ABB RobotStudio station: Second Assignment.rspag

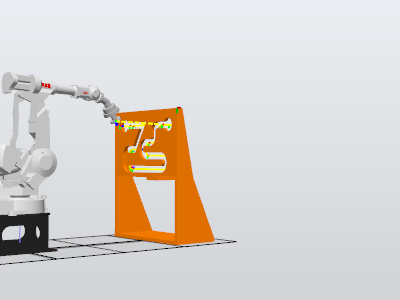
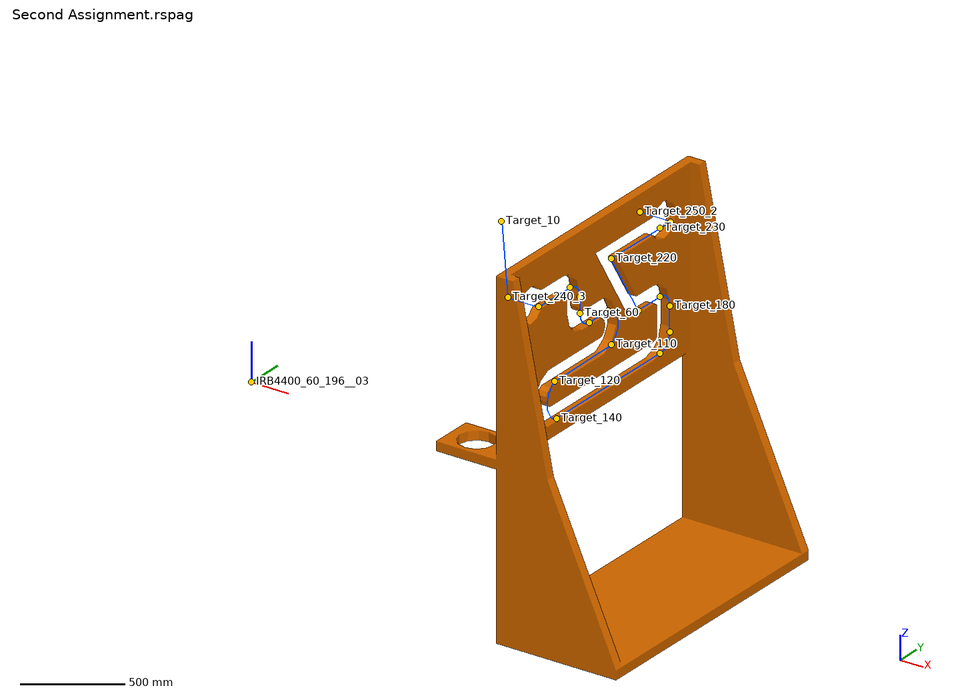
[picture v1: parts stored in the station drawn from their meshes, with robot base, taught points and paths (robot models come from the ABB library and are not in the file)]
--- station ---
Station station (saved by RobotStudio 24.1.10713.1)
Controller Controller3, task T_ROB1: task frame (RAPID world) sits at (0, 0, 500.21) mm in the station
Controller Controller3
  mechanical unit ROB_1: IRB4400_60_196__03, 6 joints, base frame (0, 0, 0) mm
Layout (positions relative to the parent item):
  - IRB4400_60_196__03 [mechanism, from %ABB.RobotStudio.Models.IRB4400%\IRB4400_60_196_G_03.rslib] at (0, 0, 500.21) mm; joint values [0.0465, 0.0523, 0.046, 0.1259, 0.3531, 3.0285] (rad or m)
  - Robotfot_IRB4400 [part, from assignment 2\Robotfot_IRB4400.rslib]
  - Tool [mechanism, from Module 2\Tool.rslib] at (1259.88, 64.75, 2124.37) mm, rotated rx -176.81 ry -67.27 rz 1.91 deg
  - tavla [part] at (2055.32, 720.6, 956.8) mm, rotated rx 90 ry 0 rz -90 deg, size 1600 x 1950 x 1050 mm
  - Part_1 [part] at (2055.32, 720.6, 956.8) mm, rotated rx 90 ry 0 rz -90 deg, size 183.4 x 0 x 50 mm
Attachment: Tool is attached to IRB4400_60_196__03 / Link6
Attachment: Workobject_1 is attached to tavla
Collision set CollisionSet_1: Tool against tavla, near miss 0 m

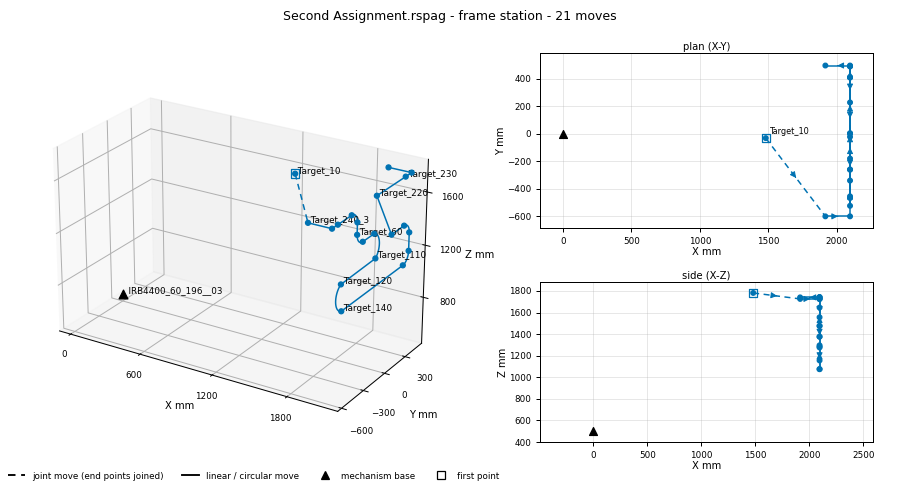
[picture p0: tool path of Second Assignment.rspag in frame station, 21 of 21 moves have a stored position in this frame; points joined in program order, loops and branches not executed]
--- Backups/Controller3/RAPID/TASK1/PROGMOD/CalibData.mod ---
MODULE CalibData
    PERS tooldata Tool:=[TRUE,[[-182.609,0,426.056],[0.958187841,0,-0.286139935,0]],[1,[0,0,1],[1,0,0,0],0,0,0]];
    TASK PERS wobjdata Workobject_1:=[FALSE,TRUE,"",[[2005.321,-829.399720938,1456.591],[0.5,-0.5,0.5,-0.5]],[[0,0,0],[1,0,0,0]]];
ENDMODULE

--- Backups/Controller3/RAPID/TASK1/PROGMOD/Module1.mod ---
MODULE Module1
        CONST robtarget Target_10:=[[-798.050043049,175.415127785,-525.051060351],[0.538949517,-0.371148696,-0.367689139,-0.660747122],[0,-1,1,0],[9E+09,9E+09,9E+09,9E+09,9E+09,9E+09]];
    CONST robtarget Target_20:=[[-306.021800708,230.811964394,89.999518831],[1,0,0,0.000000001],[-1,0,2,0],[9E+09,9E+09,9E+09,9E+09,9E+09,9E+09]];
    CONST robtarget Target_30:=[[-489.41926033,230.811964394,89.999518831],[1,0,0,0.000000001],[-1,0,2,0],[9E+09,9E+09,9E+09,9E+09,9E+09,9E+09]];
    CONST robtarget Target_40:=[[-545.987802787,254.243421862,89.999518831],[1,0,0,0.000000001],[-1,0,2,0],[9E+09,9E+09,9E+09,9E+09,9E+09,9E+09]];
    CONST robtarget Target_50:=[[-569.41926033,310.811964393,89.999518831],[1,0,0,0.000000001],[-1,0,2,0],[9E+09,9E+09,9E+09,9E+09,9E+09,9E+09]];
    CONST robtarget Target_60:=[[-569.41926033,400.811964393,89.999518831],[1,0,0,0.000000001],[-1,0,2,0],[9E+09,9E+09,9E+09,9E+09,9E+09,9E+09]];
    CONST robtarget Target_70:=[[-592.850717797,457.380506852,89.999518831],[1,0,0,0.000000001],[-1,0,2,0],[9E+09,9E+09,9E+09,9E+09,9E+09,9E+09]];
    CONST robtarget Target_80:=[[-649.41926033,480.811964394,89.999518831],[1,0,0,0.000000001],[-1,0,2,0],[9E+09,9E+09,9E+09,9E+09,9E+09,9E+09]];
    CONST robtarget Target_90:=[[-807.406978952,480.811964394,89.999518831],[1,0,0,0.000000001],[0,0,2,0],[9E+09,9E+09,9E+09,9E+09,9E+09,9E+09]];
    CONST robtarget Target_100:=[[-885.138458405,580.811964394,89.999518831],[1,0,0,0.000000001],[0,0,2,0],[9E+09,9E+09,9E+09,9E+09,9E+09,9E+09]];
    CONST robtarget Target_110:=[[-833.882147816,673.227355865,89.999518831],[1,0,0,0.000000001],[0,0,2,0],[9E+09,9E+09,9E+09,9E+09,9E+09,9E+09]];
    CONST robtarget Target_120:=[[-362.535900123,680.811964394,89.999518831],[1,0,0,0.000000001],[-1,0,2,0],[9E+09,9E+09,9E+09,9E+09,9E+09,9E+09]];
    CONST robtarget Target_130:=[[-295.929904216,780.811964394,89.999518831],[1,0,0,0.000000001],[-1,0,2,0],[9E+09,9E+09,9E+09,9E+09,9E+09,9E+09]];
    CONST robtarget Target_140:=[[-374.868021865,882.356636788,89.999518831],[1,0,0,0.000000001],[-1,0,2,0],[9E+09,9E+09,9E+09,9E+09,9E+09,9E+09]];
    CONST robtarget Target_150:=[[-1239.41926033,880.811964394,89.999518831],[1,0,0,0.000000001],[0,0,2,0],[9E+09,9E+09,9E+09,9E+09,9E+09,9E+09]];
    CONST robtarget Target_160:=[[-1295.987802862,857.380506852,89.999518831],[1,0,0,0.000000001],[0,0,2,0],[9E+09,9E+09,9E+09,9E+09,9E+09,9E+09]];
    CONST robtarget Target_170:=[[-1319.41926033,800.811964393,89.999518831],[1,0,0,0.000000001],[0,0,2,0],[9E+09,9E+09,9E+09,9E+09,9E+09,9E+09]];
    CONST robtarget Target_180:=[[-1319.41926033,660.811964393,89.999518831],[1,0,0,0.000000001],[0,0,2,0],[9E+09,9E+09,9E+09,9E+09,9E+09,9E+09]];
    CONST robtarget Target_190:=[[-1295.987802862,604.243421935,89.999518831],[1,0,0,0.000000001],[0,0,2,0],[9E+09,9E+09,9E+09,9E+09,9E+09,9E+09]];
    CONST robtarget Target_200:=[[-1239.41926033,580.811964394,89.999518831],[1,0,0,0.000000001],[0,0,2,0],[9E+09,9E+09,9E+09,9E+09,9E+09,9E+09]];
    CONST robtarget Target_210:=[[-1057.306096355,580.811964393,89.999518831],[1,0,0,0.000000001],[0,0,2,0],[9E+09,9E+09,9E+09,9E+09,9E+09,9E+09]];
    CONST robtarget Target_220:=[[-830.471485674,212.952696239,89.999518831],[1,0,0,0.000000001],[0,0,2,0],[9E+09,9E+09,9E+09,9E+09,9E+09,9E+09]];
    CONST robtarget Target_230:=[[-1239.034176521,216.505554326,89.999518831],[1,0,0,0.000000001],[0,0,2,0],[9E+09,9E+09,9E+09,9E+09,9E+09,9E+09]];
    CONST robtarget Target_240:=[[-229.419720938,230.812241944,90],[1,0,0,0.000000001],[-1,0,2,0],[9E+09,9E+09,9E+09,9E+09,9E+09,9E+09]];
    CONST robtarget Target_250:=[[-1325.636720938,216.505241944,90],[0.996194698,0,0,-0.087155742],[0,0,2,0],[9E+09,9E+09,9E+09,9E+09,9E+09,9E+09]];
    CONST robtarget Target_260:=[[-828.754222431,730.811964394,49.999518831],[0.866025404,0,0,0.5],[0,-2,1,0],[9E+09,9E+09,9E+09,9E+09,9E+09,9E+09]];
    CONST robtarget Target_270:=[[-378.327740435,730.811964394,49.999518831],[0.866025404,0,0,0.5],[-1,-2,1,0],[9E+09,9E+09,9E+09,9E+09,9E+09,9E+09]];
    CONST robtarget Target_280:=[[-378.327740435,730.811964394,-0.000481169],[0.866025404,0,0,0.5],[-1,-2,1,0],[9E+09,9E+09,9E+09,9E+09,9E+09,9E+09]];
    CONST robtarget Target_290:=[[-349.904940542,760.32494624,-0.000481169],[0.866025404,0,0,0.5],[-1,-2,1,0],[9E+09,9E+09,9E+09,9E+09,9E+09,9E+09]];
    CONST robtarget Target_300:=[[-349.904940542,801.298982547,-0.000481169],[0.866025404,0,0,0.5],[-1,-2,1,0],[9E+09,9E+09,9E+09,9E+09,9E+09,9E+09]];
    CONST robtarget Target_310:=[[-378.327740435,830.811964394,-0.000481169],[0.866025404,0,0,0.5],[-1,-2,1,0],[9E+09,9E+09,9E+09,9E+09,9E+09,9E+09]];
    CONST robtarget Target_320:=[[-349.904940542,760.32494624,-0.000481169],[0.866025404,0,0,0.5],[-1,-2,1,0],[9E+09,9E+09,9E+09,9E+09,9E+09,9E+09]];
    CONST robtarget Target_330:=[[-349.904940542,801.298982547,-0.000481169],[0.866025404,0,0,0.5],[-1,-2,1,0],[9E+09,9E+09,9E+09,9E+09,9E+09,9E+09]];
    CONST robtarget Target_340:=[[-378.327740435,830.811964394,-0.000481169],[0.866025404,0,0,0.5],[-1,-2,1,0],[9E+09,9E+09,9E+09,9E+09,9E+09,9E+09]];
    CONST robtarget Target_350:=[[-1239.41926033,830.811964394,-0.000481169],[0.866025404,0,0,0.5],[0,-2,1,0],[9E+09,9E+09,9E+09,9E+09,9E+09,9E+09]];
    CONST robtarget Target_360:=[[-1254.41926033,826.792726507,-0.000481169],[0.866025404,0,0,0.5],[0,-2,1,0],[9E+09,9E+09,9E+09,9E+09,9E+09,9E+09]];
    CONST robtarget Target_370:=[[-1265.400022443,815.811964393,-0.000481169],[0.866025404,0,0,0.5],[0,-2,1,0],[9E+09,9E+09,9E+09,9E+09,9E+09,9E+09]];
    CONST robtarget Target_380:=[[-1269.41926033,800.811964393,-0.000481169],[0.866025404,0,0,0.5],[0,-2,1,0],[9E+09,9E+09,9E+09,9E+09,9E+09,9E+09]];
    CONST robtarget Target_390:=[[-1269.41926033,660.811964393,-0.000481169],[0.866025404,0,0,0.5],[0,-2,0,0],[9E+09,9E+09,9E+09,9E+09,9E+09,9E+09]];
    CONST robtarget Target_400:=[[-1265.400022443,645.811964393,-0.000481169],[0.866025404,0,0,0.5],[0,-2,0,0],[9E+09,9E+09,9E+09,9E+09,9E+09,9E+09]];
    CONST robtarget Target_410:=[[-1254.41926033,634.83120228,-0.000481169],[0.866025404,0,0,0.5],[0,-2,0,0],[9E+09,9E+09,9E+09,9E+09,9E+09,9E+09]];
    CONST robtarget Target_420:=[[-1239.41926033,630.811964394,-0.000481169],[0.866025404,0,0,0.5],[0,-2,0,0],[9E+09,9E+09,9E+09,9E+09,9E+09,9E+09]];
    CONST robtarget Target_430:=[[-1041.532424304,630.811964393,-0.000481169],[0.866025404,0,0,0.5],[0,-2,0,0],[9E+09,9E+09,9E+09,9E+09,9E+09,9E+09]];
    CONST robtarget Target_440:=[[-754.771227196,166.505554326,-0.000481169],[0.866025404,0,0,0.5],[0,-1,0,0],[9E+09,9E+09,9E+09,9E+09,9E+09,9E+09]];
    CONST robtarget Target_450:=[[-1239.034176521,166.505554326,-0.000481169],[0.866025404,0,0,0.5],[0,-1,0,0],[9E+09,9E+09,9E+09,9E+09,9E+09,9E+09]];
    CONST robtarget Target_460:=[[-1280.756798879,127.142290293,-0.000481169],[0.866025404,0,0,0.5],[0,-1,0,0],[9E+09,9E+09,9E+09,9E+09,9E+09,9E+09]];
    CONST robtarget Target_470:=[[-1337.246008312,117.181718551,-0.000481169],[0.866025404,0,0,0.5],[0,-1,0,0],[9E+09,9E+09,9E+09,9E+09,9E+09,9E+09]];
    CONST robtarget Target_480:=[[-1389.915477868,139.901110014,-0.000481169],[0.866025404,0,0,0.5],[0,-1,0,0],[9E+09,9E+09,9E+09,9E+09,9E+09,9E+09]];
    CONST robtarget Target_490:=[[-1421.435668131,187.825231055,-0.000481169],[0.866025404,0,0,0.5],[0,-1,0,0],[9E+09,9E+09,9E+09,9E+09,9E+09,9E+09]];
    CONST robtarget Target_500:=[[-1421.435668131,245.185877597,-0.000481169],[0.866025404,0,0,0.5],[0,-1,0,0],[9E+09,9E+09,9E+09,9E+09,9E+09,9E+09]];
    CONST robtarget Target_510:=[[-1389.915477868,293.109998638,-0.000481169],[0.866025404,0,0,0.5],[0,-1,0,0],[9E+09,9E+09,9E+09,9E+09,9E+09,9E+09]];
    CONST robtarget Target_520:=[[-1337.246008311,315.8293901,-0.000481169],[0.866025404,0,0,0.5],[0,-1,0,0],[9E+09,9E+09,9E+09,9E+09,9E+09,9E+09]];
    CONST robtarget Target_530:=[[-1280.756798879,305.868818358,-0.000481169],[0.866025404,0,0,0.5],[0,-1,0,0],[9E+09,9E+09,9E+09,9E+09,9E+09,9E+09]];
    CONST robtarget Target_540:=[[-1239.034176521,266.505554326,-0.000481169],[0.866025404,0,0,0.5],[0,-1,0,0],[9E+09,9E+09,9E+09,9E+09,9E+09,9E+09]];
    CONST robtarget Target_550:=[[-934.067293463,266.505554325,-0.000481169],[0.866025404,0,0,0.5],[0,-1,0,0],[9E+09,9E+09,9E+09,9E+09,9E+09,9E+09]];
    CONST robtarget Target_560:=[[-934.067293463,266.505554325,49.999518831],[0.866025404,0,0,0.5],[0,-1,0,0],[9E+09,9E+09,9E+09,9E+09,9E+09,9E+09]];
    CONST robtarget Target_570:=[[-1097.306096355,530.811964393,49.999518831],[0.866025404,0,0,0.5],[0,-2,0,0],[9E+09,9E+09,9E+09,9E+09,9E+09,9E+09]];
    CONST robtarget Target_580:=[[-1239.41926033,530.811964394,49.999518831],[0.866025404,0,0,0.5],[0,-1,0,0],[9E+09,9E+09,9E+09,9E+09,9E+09,9E+09]];
    CONST robtarget Target_590:=[[-1304.41926033,548.228661902,49.999518831],[0.866025404,0,0,0.5],[0,-1,0,0],[9E+09,9E+09,9E+09,9E+09,9E+09,9E+09]];
    CONST robtarget Target_600:=[[-1352.002562822,595.811964394,49.999518831],[0.866025404,0,0,0.5],[0,-1,0,0],[9E+09,9E+09,9E+09,9E+09,9E+09,9E+09]];
    CONST robtarget Target_610:=[[-1369.41926033,660.811964393,49.999518831],[0.866025404,0,0,0.5],[0,-2,0,0],[9E+09,9E+09,9E+09,9E+09,9E+09,9E+09]];
    CONST robtarget Target_620:=[[-1369.41926033,800.811964393,49.999518831],[0.866025404,0,0,0.5],[0,-2,1,0],[9E+09,9E+09,9E+09,9E+09,9E+09,9E+09]];
    CONST robtarget Target_630:=[[-1352.002562822,865.811964393,49.999518831],[0.866025404,0,0,0.5],[0,-2,1,0],[9E+09,9E+09,9E+09,9E+09,9E+09,9E+09]];
    CONST robtarget Target_640:=[[-1304.41926033,913.395266885,49.999518831],[0.866025404,0,0,0.5],[0,-2,1,0],[9E+09,9E+09,9E+09,9E+09,9E+09,9E+09]];
    CONST robtarget Target_650:=[[-1239.41926033,930.811964393,49.999518831],[0.866025404,0,0,0.5],[0,-2,1,0],[9E+09,9E+09,9E+09,9E+09,9E+09,9E+09]];
    CONST robtarget Target_660:=[[-362.535900123,930.811964394,49.999518831],[0.866025404,0,0,0.5],[-1,-2,1,0],[9E+09,9E+09,9E+09,9E+09,9E+09,9E+09]];
    CONST robtarget Target_670:=[[-302.218171068,900.212228118,49.999518831],[0.866025404,0,0,0.5],[-1,-2,1,0],[9E+09,9E+09,9E+09,9E+09,9E+09,9E+09]];
    CONST robtarget Target_680:=[[-260.707397504,846.813464306,49.999518831],[0.866025404,0,0,0.5],[-1,-3,1,0],[9E+09,9E+09,9E+09,9E+09,9E+09,9E+09]];
    CONST robtarget Target_690:=[[-245.929904216,780.811964394,49.999518831],[0.866025404,0,0,0.5],[-1,-3,1,0],[9E+09,9E+09,9E+09,9E+09,9E+09,9E+09]];
    CONST robtarget Target_700:=[[-260.707397504,714.810464481,49.999518831],[0.866025404,0,0,0.5],[-1,-3,1,0],[9E+09,9E+09,9E+09,9E+09,9E+09,9E+09]];
    CONST robtarget Target_710:=[[-302.218171068,661.411700669,49.999518831],[0.866025404,0,0,0.5],[-1,-2,1,0],[9E+09,9E+09,9E+09,9E+09,9E+09,9E+09]];
    CONST robtarget Target_720:=[[-362.535900123,630.811964394,49.999518831],[0.866025404,0,0,0.5],[-1,-2,1,0],[9E+09,9E+09,9E+09,9E+09,9E+09,9E+09]];
    CONST robtarget Target_730:=[[-807.406978952,630.811964394,49.999518831],[0.866025404,0,0,0.5],[0,-2,1,0],[9E+09,9E+09,9E+09,9E+09,9E+09,9E+09]];
    CONST robtarget Target_740:=[[-831.811504771,600.334219668,49.999518831],[0.866025404,0,0,0.5],[0,-2,0,0],[9E+09,9E+09,9E+09,9E+09,9E+09,9E+09]];
    CONST robtarget Target_750:=[[-831.811504771,561.289709119,49.999518831],[0.866025404,0,0,0.5],[0,-2,0,0],[9E+09,9E+09,9E+09,9E+09,9E+09,9E+09]];
    CONST robtarget Target_760:=[[-807.406978952,530.811964393,49.999518831],[0.866025404,0,0,0.5],[0,-2,0,0],[9E+09,9E+09,9E+09,9E+09,9E+09,9E+09]];
    CONST robtarget Target_770:=[[-649.41926033,530.811964394,49.999518831],[0.866025404,0,0,0.5],[-1,-2,0,0],[9E+09,9E+09,9E+09,9E+09,9E+09,9E+09]];
    CONST robtarget Target_780:=[[-584.41926033,513.395266885,49.999518831],[0.866025404,0,0,0.5],[-1,-2,0,0],[9E+09,9E+09,9E+09,9E+09,9E+09,9E+09]];
    CONST robtarget Target_790:=[[-536.835957838,465.811964393,49.999518831],[0.866025404,0,0,0.5],[-1,-2,0,0],[9E+09,9E+09,9E+09,9E+09,9E+09,9E+09]];
    CONST robtarget Target_800:=[[-519.41926033,400.811964393,49.999518831],[0.866025404,0,0,0.5],[-1,-1,0,0],[9E+09,9E+09,9E+09,9E+09,9E+09,9E+09]];
    CONST robtarget Target_810:=[[-519.41926033,310.811964393,49.999518831],[0.866025404,0,0,0.5],[-1,-1,0,0],[9E+09,9E+09,9E+09,9E+09,9E+09,9E+09]];
    CONST robtarget Target_820:=[[-515.400022443,295.811964393,49.999518831],[0.866025404,0,0,0.5],[-1,-1,0,0],[9E+09,9E+09,9E+09,9E+09,9E+09,9E+09]];
    CONST robtarget Target_830:=[[-504.41926033,284.83120228,49.999518831],[0.866025404,0,0,0.5],[-1,-1,0,0],[9E+09,9E+09,9E+09,9E+09,9E+09,9E+09]];
    CONST robtarget Target_840:=[[-489.41926033,280.811964393,49.999518831],[0.866025404,0,0,0.5],[-1,-1,0,0],[9E+09,9E+09,9E+09,9E+09,9E+09,9E+09]];
    CONST robtarget Target_850:=[[-306.021800708,280.811964394,49.999518831],[0.866025404,0,0,0.5],[-1,-1,-1,0],[9E+09,9E+09,9E+09,9E+09,9E+09,9E+09]];
    CONST robtarget Target_860:=[[-264.29917835,320.175228426,49.999518831],[0.866025404,0,0,0.5],[-1,0,-1,0],[9E+09,9E+09,9E+09,9E+09,9E+09,9E+09]];
    CONST robtarget Target_870:=[[-207.809968917,330.135800168,49.999518831],[0.866025404,0,0,0.5],[-1,0,-1,0],[9E+09,9E+09,9E+09,9E+09,9E+09,9E+09]];
    CONST robtarget Target_880:=[[-155.140499361,307.416408705,49.999518831],[0.866025404,0,0,0.5],[-1,0,-1,0],[9E+09,9E+09,9E+09,9E+09,9E+09,9E+09]];
    CONST robtarget Target_890:=[[-123.620309098,259.492287665,49.999518831],[0.866025404,0,0,0.5],[-1,0,-1,0],[9E+09,9E+09,9E+09,9E+09,9E+09,9E+09]];
    CONST robtarget Target_900:=[[-123.620309098,202.131641122,49.999518831],[0.866025404,0,0,0.5],[-1,0,-1,0],[9E+09,9E+09,9E+09,9E+09,9E+09,9E+09]];
    CONST robtarget Target_910:=[[-155.140499361,154.207520082,49.999518831],[0.866025404,0,0,0.5],[-1,0,-1,0],[9E+09,9E+09,9E+09,9E+09,9E+09,9E+09]];
    CONST robtarget Target_920:=[[-207.809968917,131.488128619,49.999518831],[0.866025404,0,0,0.5],[-1,0,-1,0],[9E+09,9E+09,9E+09,9E+09,9E+09,9E+09]];
    CONST robtarget Target_930:=[[-264.29917835,141.448700361,49.999518831],[0.866025404,0,0,0.5],[-1,0,-1,0],[9E+09,9E+09,9E+09,9E+09,9E+09,9E+09]];
    CONST robtarget Target_940:=[[-306.021800708,180.811964394,49.999518831],[0.866025404,0,0,0.5],[-1,-1,-1,0],[9E+09,9E+09,9E+09,9E+09,9E+09,9E+09]];
    CONST robtarget Target_250_2:=[[-1325.636720938,216.505241944,-90],[0.996194698,0,0,-0.087155742],[0,0,2,0],[9E+09,9E+09,9E+09,9E+09,9E+09,9E+09]];
    CONST robtarget Target_240_3:=[[-229.419720938,230.812241944,-90],[1,0,0,0.000000001],[-1,0,2,0],[9E+09,9E+09,9E+09,9E+09,9E+09,9E+09]];
!***********************************************************
    !
    ! Module:  Module1
    !
    ! Description:
    !   <Insert description here>
    !
    ! Author: haba0028
    !
    ! Version: 1.0
    !
    !***********************************************************


    !***********************************************************
    !
    ! Procedure main
    !
    !   This is the entry point of your program
    !
    !***********************************************************
    PROC main()
        !Add your code here
        Path_10;
    ENDPROC
    PROC Path_10()
        MoveJ Target_10,v1000,fine,Tool\WObj:=Workobject_1;
        MoveJ Target_240_3,v1000,fine,Tool\WObj:=Workobject_1;
        MoveL Target_240,v1000,fine,Tool\WObj:=Workobject_1;
        MoveL Target_20,v1000,fine,Tool\WObj:=Workobject_1;
        MoveL Target_30,v1000,fine,Tool\WObj:=Workobject_1;
        MoveC Target_40,Target_50,v1000,fine,Tool\WObj:=Workobject_1;
        MoveL Target_60,v1000,fine,Tool\WObj:=Workobject_1;
        MoveC Target_70,Target_80,v1000,fine,Tool\WObj:=Workobject_1;
        MoveL Target_90,v1000,fine,Tool\WObj:=Workobject_1;
        MoveC Target_100,Target_110,v1000,fine,Tool\WObj:=Workobject_1;
        MoveL Target_120,v1000,fine,Tool\WObj:=Workobject_1;
        MoveC Target_130,Target_140,v1000,fine,Tool\WObj:=Workobject_1;
        MoveL Target_150,v1000,fine,Tool\WObj:=Workobject_1;
        MoveC Target_160,Target_170,v1000,fine,Tool\WObj:=Workobject_1;
        MoveL Target_180,v1000,fine,Tool\WObj:=Workobject_1;
        MoveC Target_190,Target_200,v1000,fine,Tool\WObj:=Workobject_1;
        MoveL Target_210,v1000,fine,Tool\WObj:=Workobject_1;
        MoveL Target_220,v1000,fine,Tool\WObj:=Workobject_1;
        MoveL Target_230,v1000,fine,Tool\WObj:=Workobject_1;
        MoveL Target_250,v1000,fine,Tool\WObj:=Workobject_1;
        MoveL Target_250_2,v1000,fine,Tool\WObj:=Workobject_1;
    ENDPROC
ENDMODULE
